// TIA Portal V16 export
// export: Created 2024-05-10T06:46:40.6574132Z, ExportSetting WithDefaults, DisplayName Totally Integrated Automation Portal, DisplayVersion V16, DisplayName TIA Portal Version Control Interface, DisplayVersion V16, DisplayName TIA Portal Openness, DisplayVersion V16, DisplayName STEP 7 Professional, DisplayVersion V16, DisplayName STEP 7 Safety, DisplayVersion V16, DisplayName WinCC Professional, DisplayVersion V16
FUNCTION_BLOCK "K02_初始化"   // FB2, LAD
{ S7_Optimized_Access := 'TRUE' }
VERSION : 0.1
// stored: AutoNumber false, IsIECCheckEnabled false, IsRetainMemResEnabled false, MemoryReserve 100, SetENOAutomatically false, UDAEnableTagReadback false
   VAR_TEMP
      M_Pluse : Array[1..2] of Bool;
      M_OneStep : Bool;   // 单步运行
   END_VAR
   VAR_TEMP   // added for the SCL form of the ladder/FBD networks
      _w1 : Bool;
   END_VAR
BEGIN

REGION Network 1: 初始化条件
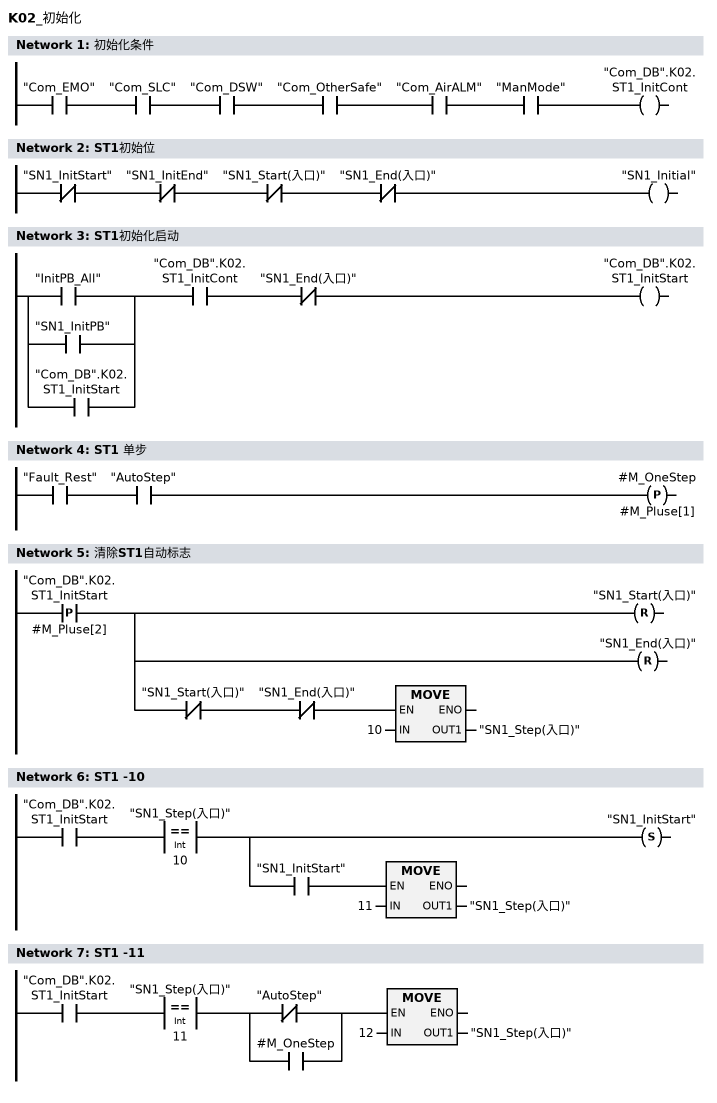
   RUNG wire#powerrail
      Contact( "Com_EMO" )
      Contact( "Com_SLC" )
      Contact( "Com_DSW" )
      Contact( "Com_OtherSafe" )
      Contact( "Com_AirALM" )
      Contact( "ManMode" )
      Coil( "Com_DB".K02.ST1_InitCont )
   END_RUNG
   // the same network as SCL:
   "Com_DB".K02.ST1_InitCont := "Com_EMO" AND "Com_SLC" AND "Com_DSW" AND "Com_OtherSafe" AND "Com_AirALM" AND "ManMode";
END_REGION

REGION Network 2: ST1初始位
   RUNG wire#powerrail
      I_Contact( "SN1_InitStart" )
      I_Contact( "SN1_InitEnd" )
      I_Contact( "SN1_Start(入口)" )
      I_Contact( "SN1_End(入口)" )
      Coil( "SN1_Initial" )
   END_RUNG
   // the same network as SCL:
   "SN1_Initial" := NOT "SN1_InitStart" AND NOT "SN1_InitEnd" AND NOT "SN1_Start(入口)" AND NOT "SN1_End(入口)";
END_REGION

REGION Network 3: ST1初始化启动
   RUNG wire#powerrail
      Contact( "InitPB_All" )
      wire#w1
      Contact( "Com_DB".K02.ST1_InitCont )
      I_Contact( "SN1_End(入口)" )
      Coil( "Com_DB".K02.ST1_InitStart )
   END_RUNG
   RUNG wire#powerrail
      Contact( "SN1_InitPB" )
   END_RUNG wire#w1
   RUNG wire#powerrail
      Contact( "Com_DB".K02.ST1_InitStart )
   END_RUNG wire#w1
   // the same network as SCL:
   "Com_DB".K02.ST1_InitStart := ("InitPB_All" OR "SN1_InitPB" OR "Com_DB".K02.ST1_InitStart) AND "Com_DB".K02.ST1_InitCont AND NOT "SN1_End(入口)";
END_REGION

REGION Network 4: ST1 单步
   #_w1 := "Fault_Rest" AND "AutoStep";
   #M_OneStep := #_w1 AND NOT #M_Pluse[1];   // rising edge
   #M_Pluse[1] := #_w1;
END_REGION

REGION Network 5: 清除ST1自动标志
   RUNG wire#powerrail
      P_Contact(operand := "Com_DB".K02.ST1_InitStart, bit := #M_Pluse[2])
      wire#w1
      R_Coil( "SN1_Start(入口)" )
   END_RUNG
   RUNG wire#w1
      R_Coil( "SN1_End(入口)" )
   END_RUNG
   RUNG wire#w1
      I_Contact( "SN1_Start(入口)" )
      I_Contact( "SN1_End(入口)" )
      Move(in := 10, out1 => "SN1_Step(入口)")
   END_RUNG
   // the same network as SCL:
   #_w1 := "Com_DB".K02.ST1_InitStart AND NOT #M_Pluse[2];   // rising edge of "Com_DB".K02.ST1_InitStart
   #M_Pluse[2] := "Com_DB".K02.ST1_InitStart;
   IF #_w1 THEN
       "SN1_Start(入口)" := FALSE;
       "SN1_End(入口)" := FALSE;
   END_IF;
   IF #_w1 AND NOT "SN1_Start(入口)" AND NOT "SN1_End(入口)" THEN "SN1_Step(入口)" := 10; END_IF;
END_REGION

REGION Network 6: ST1 -10
   RUNG wire#powerrail
      Contact( "Com_DB".K02.ST1_InitStart )
      { S7_Templates := "SrcType := Int" } EQ_Contact(in1 := "SN1_Step(入口)", in2 := 10)
      wire#w1
      S_Coil( "SN1_InitStart" )
   END_RUNG
   RUNG wire#w1
      Contact( "SN1_InitStart" )
      Move(in := 11, out1 => "SN1_Step(入口)")
   END_RUNG
   // the same network as SCL:
   #_w1 := "Com_DB".K02.ST1_InitStart AND ("SN1_Step(入口)" = 10);
   IF #_w1 THEN "SN1_InitStart" := TRUE; END_IF;
   IF #_w1 AND "SN1_InitStart" THEN "SN1_Step(入口)" := 11; END_IF;
END_REGION

REGION Network 7: ST1 -11
   RUNG wire#powerrail
      Contact( "Com_DB".K02.ST1_InitStart )
      { S7_Templates := "SrcType := Int" } EQ_Contact(in1 := "SN1_Step(入口)", in2 := 11)
      wire#w1
      I_Contact( "AutoStep" )
      wire#w2
      Move(in := 12, out1 => "SN1_Step(入口)")
   END_RUNG
   RUNG wire#w1
      Contact( #M_OneStep )
   END_RUNG wire#w2
   // the same network as SCL:
   IF "Com_DB".K02.ST1_InitStart AND ("SN1_Step(入口)" = 11) AND (NOT "AutoStep" OR #M_OneStep) THEN
       "SN1_Step(入口)" := 12;
   END_IF;
END_REGION
END_FUNCTION_BLOCK
